// TIA Portal project "Profizumo" (V17)

(* hardware
DEVICE "S7-1500/ET200MP-Station_1"  S7-1500 station
   slot 0: "Profilschiene_0"  Rack  6ES7 590-1***0-0AA0
   slot 1: "PLC_1"  CPU 1516-3 PN/DP  6ES7 516-3AN01-0AB0  V2.9
      slot 3: "CPU-Display_1"  6ES7591-1BA00-0AA0
      slot 32768: "PROFINET-Schnittstelle_1"  X1
      slot 33024: "PROFINET-Schnittstelle_2"  X2
      slot 33280: "DP-Schnittstelle_1"  X3
      slot 34817: "Virtual CP interface port_1"  Virtual CP interface port  Virtual CP interface port
DEVICE "S7-1500/ET200MP-Station_2"  S7-1500 station
   slot 0: "Profilschiene_0"  Rack  6ES7 590-1***0-0AA0
   slot 1: "workstation3.rio"  IM 155-5 PN ST  6ES7 155-5AA01-0AB0  V4.1
   slot 2: "DI 32x24VDC HF_1"  DI 32x24VDC HF  6ES7 521-1BL00-0AB0  V2.1
   slot 3: "DQ 32x24VDC/0.5A ST_1"  DQ 32x24VDC/0.5A ST  6ES7 522-1BL00-0AB0  V2.0
   slot 4: "AI 8xU/I/RTD/TC ST_1"  AI 8xU/I/RTD/TC ST  6ES7 531-7KF00-0AB0  V2.0
   slot 5: "AQ 4xU/I ST_1"  AQ 4xU/I ST  6ES7 532-5HD00-0AB0  V2.0
DEVICE "GSD-Geraet_1"  GSD.Device.PN
   slot 0: "Baugruppenträger"  Rack  V1.0
   slot 0: "profizumo"  Profizumo  123 444 555  V0.1.1
      slot 0: "Profizumo"  Profizumo
      slot 1: "X1"  X1
         slot 1: "X1 P1"  X1 P1
      slot 1: "Motors_1"  Motors  1.0
         slot 0: "Motors submodule"  Motors submodule
   slot 2: "IMU sensors_1"  IMU sensors  1.0
      slot 0: "Acceleration"  Acceleration
      slot 1: "Gyro"  Gyro
      slot 2: "Magnetometer"  Magnetometer
   slot 3: "Ultrasound distance sensor_1"  Ultrasound distance sensor  1.0
      slot 0: "Ultrasound distance sensor"  Ultrasound distance sensor
*)

// ===== PLC "PLC_1"  CPU 1516-3 PN/DP =====

VAR_GLOBAL   // PLC tag table "Standard-Variablentabelle"
   "zumoOutputs" AT %I0.0 : "typeZumoOutputs";
   "leftButton" AT %I20.0 : Bool;
   "rightButton" AT %I20.1 : Bool;
   "zumoInputs" AT %Q0.0 : "typeZumoInputs";
   "Tag_1" AT %Q4.0 : "typeZumoInputs";
END_VAR

TYPE "typeZumoOutputs"
VERSION : 0.1
   STRUCT
      accelerationX : Int;
      accelerationY : Int;
      accelerationZ : Int;
      gyroX : Int;
      gyroY : Int;
      gyroZ : Int;
      magnetometerX : Int;
      magnetometerY : Int;
      magnetometerZ : Int;
      distance_mm : Int;
   END_STRUCT;
END_TYPE

TYPE "typeZumoInputs"
VERSION : 0.1
   STRUCT
      leftMotorSpeed : Int;
      rightMotorSpeed : Int;
   END_STRUCT;
END_TYPE

ORGANIZATION_BLOCK "Main"   // OB1, LAD, ProgramCycle
TITLE = "Main Program Sweep (Cycle)"
{ S7_Optimized_Access := 'TRUE' }
VERSION : 0.1
   VAR_INPUT
      Initial_Call : Bool;   // Initial call of this OB
      Remanence : Bool;   // =True, if remanent data are available
   END_VAR
BEGIN

REGION Network 1
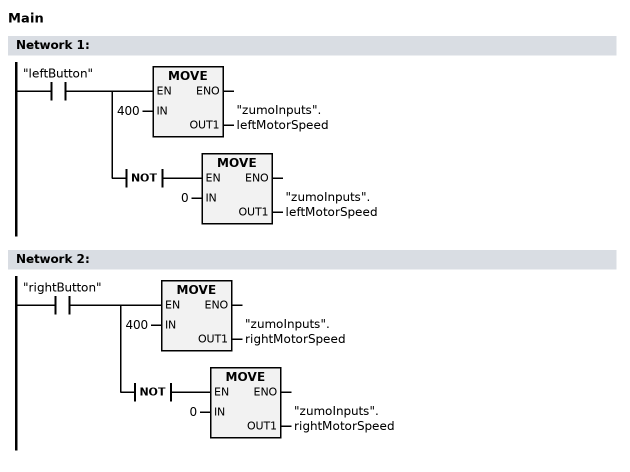
   RUNG wire#powerrail
      Contact( "leftButton" )
      wire#w1
      Move(in := 400, out1 => "zumoInputs".leftMotorSpeed)
   END_RUNG
   RUNG wire#w1
      Not()
      Move(in := 0, out1 => "zumoInputs".leftMotorSpeed)
   END_RUNG
   // the same network as SCL:
   IF "leftButton" THEN "zumoInputs".leftMotorSpeed := 400; END_IF;
   IF NOT "leftButton" THEN "zumoInputs".leftMotorSpeed := 0; END_IF;
END_REGION

REGION Network 2
   RUNG wire#powerrail
      Contact( "rightButton" )
      wire#w1
      Move(in := 400, out1 => "zumoInputs".rightMotorSpeed)
   END_RUNG
   RUNG wire#w1
      Not()
      Move(in := 0, out1 => "zumoInputs".rightMotorSpeed)
   END_RUNG
   // the same network as SCL:
   IF "rightButton" THEN "zumoInputs".rightMotorSpeed := 400; END_IF;
   IF NOT "rightButton" THEN "zumoInputs".rightMotorSpeed := 0; END_IF;
END_REGION
END_ORGANIZATION_BLOCK